   A_1942_MXZ0MA.A_1942_MXZ01.Par.ParHornCode := 0;
   A_1942_MXZ0MA.A_1942_MXZ01.Par.ParLogOff := FALSE;
   A_1942_MXZ0MA.A_1942_MXZ01.Par.ParManual := TRUE;
   A_1942_MXZ0MA.A_1942_MXZ01.Par.ParRestartDelay := FALSE;
   A_1942_MXZ0MA.A_1942_MXZ01.Par.Par2Speed := TRUE;
   A_1942_MXZ0MA.A_1942_MXZ01.Par.ParHeavyStartup := FALSE;
   A_1942_MXZ0MA.A_1942_MXZ01.Par.spare45 := FALSE;
   A_1942_MXZ0MA.A_1942_MXZ01.Par.spare46 := FALSE;
   A_1942_MXZ0MA.A_1942_MXZ01.Par.OutEdgeFaultReset := FALSE;
   A_1942_MXZ0MA.A_1942_MXZ01.Par.OutDelayFault := FALSE;
   A_1942_MXZ0MA.A_1942_MXZ01.Par.OutFlagFaultDev := FALSE;
   A_1942_MXZ0MA.A_1942_MXZ01.Par.ParMonTime := 50;
   A_1942_MXZ0MA.A_1942_MXZ01.Par.ParStartingTime := 20;
   A_1942_MXZ0MA.A_1942_MXZ01.Par.ParStoppingTime := 50;
   A_1942_MXZ0MA.A_1942_MXZ01.Par.ParIdlingTime := 0;
   A_1942_MXZ0MA.A_1942_MXZ01.Par.ParDelayTime := 10;
   A_1942_MXZ0MA.A_1942_MXZ01.Par.OutMonTime := 0;
   A_1942_MXZ0MA.A_1942_MXZ01.Par.OutTransitionTime := 0;
   A_1942_MXZ0MA.A_1942_MXZ01.Par.OutDelayTime := 0;
   A_1942_MXZ0MA.A_1942_MXZ01.Par.InOutManPulseLen := 0;
   A_1941_QXV31.StCode := 0;
   A_1941_QXV31.InEnableLN := FALSE;
   A_1941_QXV31.InEnableHN := FALSE;
   A_1941_QXV31.InStopCTime := FALSE;
   A_1941_QXV31.spare0203 := FALSE;
   A_1941_QXV31.spare0204 := FALSE;
   A_1941_QXV31.InpLN := FALSE;
   A_1941_QXV31.InpHN := FALSE;
   A_1941_QXV31.InpFaultDev := FALSE;
   A_1941_QXV31.CmdLN := FALSE;
   A_1941_QXV31.CmdHN := FALSE;
   A_1941_QXV31.CmdNext := FALSE;
   A_1941_QXV31.CmdFaultReset := FALSE;
   A_1941_QXV31.InLocal := FALSE;
   A_1941_QXV31.InManual := FALSE;
   A_1941_QXV31.InReport := FALSE;
   A_1941_QXV31.InSeqStop := FALSE;
   A_1941_QXV31.InHWStop := FALSE;
   A_1941_QXV31.InDPFault := FALSE;
   A_1941_QXV31.OutIdling := FALSE;
   A_1941_QXV31.OutDelayFault := FALSE;
   A_1941_QXV31.OutMonFault := FALSE;
   A_1941_QXV31.OutpLN := FALSE;
   A_1941_QXV31.OutpHN := FALSE;
   A_1941_QXV31.spare0407 := FALSE;
   A_1941_QXV31.StLN := FALSE;
   A_1941_QXV31.StCtoHN := FALSE;
   A_1941_QXV31.StHN := FALSE;
   A_1941_QXV31.StCtoLN := FALSE;
   A_1941_QXV31.StFault := FALSE;
   A_1941_QXV31.StNoPosition := FALSE;
   A_1941_QXV31.OutAlarmNrLog := 0;
   A_1941_QXV31.Par.ParObjectNo := 0;
   A_1941_QXV31.Par.ParMsgType := 0;
   A_1941_QXV31.Par.ParHornCode := 0;
   A_1941_QXV31.Par.ParLogOff := FALSE;
   A_1941_QXV31.Par.ParManual := TRUE;
   A_1941_QXV31.Par.ParPulseValve := FALSE;
   A_1941_QXV31.Par.ParContValve := FALSE;
   A_1941_QXV31.Par.ParManualFlap := FALSE;
   A_1941_QXV31.Par.ParMonTime := 0;
   A_1941_QXV31.Par.ParPulseTimeHN := 0;
   A_1941_QXV31.Par.ParPulseTimeLN := 0;
   A_1941_QXV31.Par.ParIdlingTime := 0;
   A_1941_QXV31.Par.ParDelayTime := 0;
   A_1941_QXV31.Par.OutMonTime := 0;
   A_1941_QXV31.Par.OutTransitionTime := 0;
   A_1941_QXV31.Par.OutDelayTime := 0;
   A_1941_QXV31.Par.InOutManPulseLen := 0;
END_DATA_BLOCK

